// TIA Portal V20 export
ORGANIZATION_BLOCK "Main"   // OB1, LAD, ProgramCycle
TITLE = "Main Program Sweep (Cycle)"
{ S7_Optimized_Access := 'TRUE' }
// stored: SetENOAutomatically false
   VAR_INPUT
      Initial_Call : Bool;   // Initial call of this OB
      Remanence : Bool;   // =True, if remanent data are available
   END_VAR
BEGIN

REGION Network 1
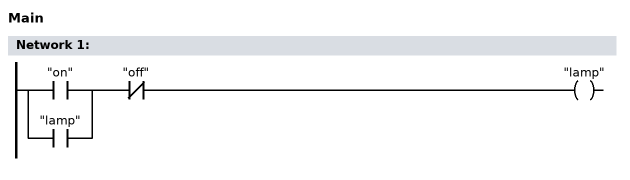
   RUNG wire#powerrail
      Contact( "on" )
      wire#w1
      I_Contact( "off" )
      Coil( "lamp" )
   END_RUNG
   RUNG wire#powerrail
      Contact( "lamp" )
   END_RUNG wire#w1
   // the same network as SCL:
   "lamp" := ("on" OR "lamp") AND NOT "off";
END_REGION
END_ORGANIZATION_BLOCK
